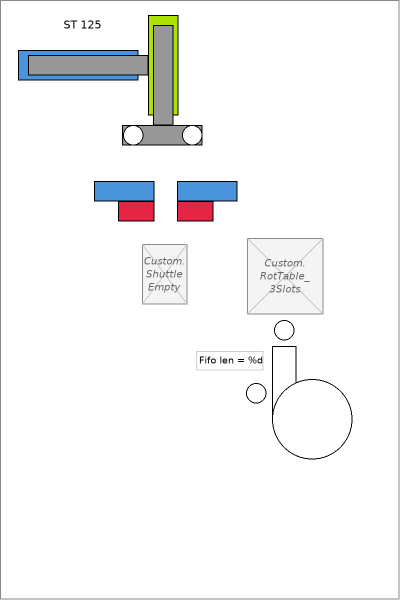
VISUALIZATION VISU_ST125  // 400x600
    Rectangle (94,181 60x20)
        p2738717112: 20*TO_INT(GVL._Process5.fb_Pnp.fb_handlingSolerohrLeft.xIN_AS)
    Rectangle (177,181 60x20)
        p2738717112: 20*TO_INT(GVL._Process5.fb_Pnp.fb_handlingSolerohrRight.xIN_AS)
    Image (142,244 45x60), invisible if: NOT __ISVALIDREF(GVL._Process5._Mover), image: Custom.Shuttle Empty
    Image (247,238 76x76), image: Custom.RotTable_3Slots
        p2858320360: ST125_Axis.axis125_10W.axis.NcToPlc.ModuloActPos
    Rectangle (18,50 120x30)
    Rectangle (28,55 120x20)
        p3560616238: GVL._Process5.fb_Pnp.fb_simu_axis125_01Y.rOUT_PixActual
    Rectangle (148,15 30x100)
        p3560616238: GVL._Process5.fb_Pnp.fb_simu_axis125_01Y.rOUT_PixActual
    Rectangle (153,25 20x100)
        p2738717112: GVL._Process5.fb_Pnp.fb_simu_axis125_02Z.rOUT_PixActual
        p3560616238: GVL._Process5.fb_Pnp.fb_simu_axis125_01Y.rOUT_PixActual
    Rectangle (272,346 24x73)
    Ellipse (272,379 80x80), colour toggle: GVL._Process5.fb_Feeder.simu_feeder.xIN_Enable
    Ellipse (246,383 20x20), colour toggle: GVL._Process5.fb_Feeder.simu_feeder.xOUT_NewPiece
    Ellipse (274,320 20x20), colour toggle: NOT GVL._Process5.fb_Feeder.simu_fifo.IsEmpty()
    Textfield (196,351 67x19), "Fifo len = %d", text variable: GVL._Process5.fb_Feeder.simu_fifo.GetLen()
    Label (40,15 85x20), "ST 125"
    Rectangle (122,125 80x20)
        p2738717112: GVL._Process5.fb_Pnp.fb_simu_axis125_02Z.rOUT_PixActual
        p3560616238: GVL._Process5.fb_Pnp.fb_simu_axis125_01Y.rOUT_PixActual
    Ellipse (123,125 20x20), colour toggle: GVL._Process5.fb_Pnp.fb_gripperFilterhutLeft.xIN_AS
        p3560616238: GVL._Process5.fb_Pnp.fb_simu_axis125_01Y.rOUT_PixActual
        p2738717112: GVL._Process5.fb_Pnp.fb_simu_axis125_02Z.rOUT_PixActual
    Ellipse (182,125 20x20), colour toggle: GVL._Process5.fb_Pnp.fb_gripperFilterhutRight.xIN_AS
        p3560616238: GVL._Process5.fb_Pnp.fb_simu_axis125_01Y.rOUT_PixActual
        p2738717112: GVL._Process5.fb_Pnp.fb_simu_axis125_02Z.rOUT_PixActual
    Rectangle (118,201 36x20), invisible if: NOT GVL._Process5.fb_Pnp.fb_gripperSolerohrLeft.xIN_AS
    Rectangle (177,201 36x20), invisible if: NOT GVL._Process5.fb_Pnp.fb_gripperSolerohrRight.xIN_AS
END_VISUALIZATION

(* stored: Version 1.1.0.1, ProductVersion 3.1.4024.6
   Visu VISU_ST125: Id {ed99920f-f9f9-4be9-a960-820d17c40ef0} *)
